// TwinCAT 3 PLC project Untitled1
// ProgramVersion: 3.1.4024.0
// libraries:
//   Tc2_Standard, * (Beckhoff Automation GmbH)
//   Tc2_System, * (Beckhoff Automation GmbH)
//   Tc3_Module, * (Beckhoff Automation GmbH)
// project tree:
//   / PlcTask.TcTTO
//   POUs/ MAIN.TcPOU
// real-time tasks:
//   TASK PlcTask: cycle T#10ms, priority 20, ADS port 350

CONFIGURATION Untitled1
    RESOURCE PLC ON TwinCAT3
        TASK PlcTask(INTERVAL := T#10ms, PRIORITY := 20);
        PROGRAM MAIN WITH PlcTask : MAIN;
    END_RESOURCE
END_CONFIGURATION

// ---- POUs/MAIN.TcPOU
PROGRAM MAIN
VAR
	fbReadIpc  : ADSREADEX := ( NETID := '192.168.3.47.1.1', PORT := 851, TMOUT := DEFAULT_ADS_TIMEOUT );
    readCommand : BOOL := FALSE;
    
    readState     : BYTE := 0;
    readBusy      : BOOL;
    readError     : BOOL;
    readErrID     : UDINT;
    countRead     : UDINT;
    
    readData   : INT;
END_VAR

CASE readState OF
    0:
        IF readCommand = TRUE THEN
            readBusy := TRUE;
            readError := FALSE;
            readErrID := 0;
            
            fbReadIpc( READ := FALSE );
            readCommand := FALSE;
            fbReadIpc( IDXGRP := 16#4040, IDXOFFS := 385008, LEN := SIZEOF(readData), DESTADDR := ADR(readData), READ := TRUE );

            readState := 1;
        END_IF
    1:
        fbReadIpc( READ := FALSE, BUSY=>readBusy, ERR=>readError, ERRID=>readErrID, COUNT_R=>countRead );
        IF readBusy = FALSE THEN
            IF readError = FALSE THEN
                readState := 0;(* Success *)
            ELSE
                readState := 100;(* Error *)
            END_IF
        END_IF
        
    100:(* TODO::Implement error handler *)
        readState := 0;
        
END_CASE

END_PROGRAM
